PROGRAM SetPosByUI
VAR
	SetPosST	: ST_SetPosByUI;
END_VAR

Axis[SetPosST.Axis].fbMC_SetPosition(
	Execute	:= SetPosST.Execute,
	Position	:= SetPosST.Position,
	Axis		:= Axis[SetPosST.Axis].Axis
);
SetPosST.Execute := FALSE;

END_PROGRAM

(* stored: Version 1.1.0.1, ProductVersion 3.1.4024.9
   POU SetPosByUI: Id {9cd913a7-d64d-4130-ae6f-5f6692c92c89}, SpecialFunc None *)
